PROGRAM MAIN
VAR
	fbPlant : PlantAndCMs.FB_PlantControl_mode_1;
	udt_plant_data_control : PlantAndCMs.Udt_PlantControl_Mode_1;
	
	fbSortingByWeight : FB_SortingByWeight;
	
	fbExitConveyors : FB_ExitSortingConveyors;
	
	fbScaleTrigger : FB_ScaleTrigger;
	fbExitLoadTrigger : FB_exitLoadTrigger;
	fbExitConveyorTrigger : FB_exitConveyorTrigger;
	
	fbWeightSorter : FB_WeightSorter;
	
	startButton : BOOL;
	
END_VAR

startButton := FALSE;

IF GVL.mb_Output_Coils[1] THEN
	startButton := TRUE;
END_IF

fbPlant(
	Ctrl_Plant := udt_plant_data_control,
	Auto_In := PlantAndCMs.FIO.bAuto,
	 
	Start_In := GVL.mb_Output_Coils[5],
	
	Stop_In := GVL.mb_Output_Coils[6],
	EmgStop_In := PlantAndCMs.FIO.bEmgStop

	);
	
	
fbSortingByWeight(
	control_data := udt_plant_data_control
	);

fbExitConveyors(
	);


fbScaleTrigger(
	scaleEntry_input := FIO2.bAtScaleEntry,
	scaleExit_input := FIO2.bAtScaleExit
		);
		
fbExitLoadTrigger(
	input_left := FIO2.bAtLeftEntry,
	input_right := FIO2.bAtRightEntry,
	input_forward := FIO2.bAtForwardEntry
	
	);
fbExitConveyorTrigger(
	inputLeft := FIO2.bAtExitLeft,
	inputRight := FIO2.bAtExitRight,
	inputForward := FIO2.bAtExitFront,	
	);
	
	
(*fbWeightSorter(
	weight_input := FIO2.rWeight,
	
	small => GVL.smallPackage,
	medium => GVL.mediumPackage,
	large => GVL.largePackage
	
	
	);*)

END_PROGRAM

(* stored: Version 1.1.0.1, ProductVersion 3.1.4024.13
   POU MAIN: Id {a7adb8ad-13f3-4f19-9d99-aac1ec4efb5e}, SpecialFunc None *)
